SUBAPPLICATION Uebung_019a (* Umschalten einer Maske *)
  (* Standard: 61499-2; Description: Copyright (c) 2023 Meisterschulen am Ostbahnhof This program and the accompanying materials are made available under the terms of the Eclipse Public License 2.0 which is available at https://www.eclipse.org/legal/epl-2.0/ SPDX-License-Identifier: EPL-2.0 *)
  (* Version 1.0, 2023-10-23, Franz Höpfinger, Meisterschulen am Ostbahnhof *)
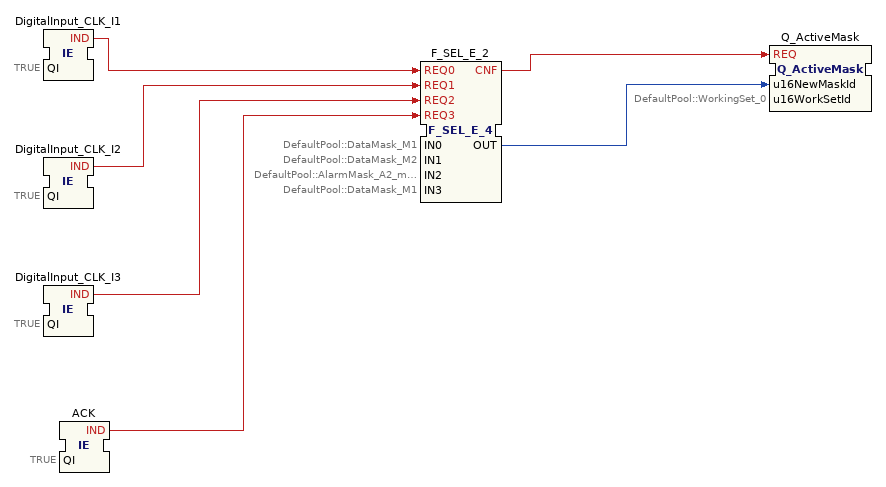
  FBS
    DigitalInput_CLK_I1 : IE(QI := TRUE);
    Q_ActiveMask : Q_ActiveMask(u16WorkSetId := DefaultPool::WorkingSet_0);
    DigitalInput_CLK_I2 : IE(QI := TRUE);
    F_SEL_E_2 : F_SEL_E_4(IN0 := DefaultPool::DataMask_M1, IN1 := DefaultPool::DataMask_M2, IN2 := DefaultPool::AlarmMask_A2_medium, IN3 := DefaultPool::DataMask_M1);
    DigitalInput_CLK_I3 : IE(QI := TRUE);
    ACK : IE(QI := TRUE);
  END_FBS
  EVENT_CONNECTIONS
    DigitalInput_CLK_I1.IND TO F_SEL_E_2.REQ0;
    DigitalInput_CLK_I2.IND TO F_SEL_E_2.REQ1;
    F_SEL_E_2.CNF TO Q_ActiveMask.REQ;
    DigitalInput_CLK_I3.IND TO F_SEL_E_2.REQ2;
    ACK.IND TO F_SEL_E_2.REQ3;
  END_CONNECTIONS
  DATA_CONNECTIONS
    F_SEL_E_2.OUT TO Q_ActiveMask.u16NewMaskId;
  END_CONNECTIONS
END_SUBAPPLICATION
